// TIA Portal V17 export
// export: Created 2023-02-13T11:16:15.1226472Z, ExportSetting WithDefaults, DisplayName Totally Integrated Automation Portal, DisplayVersion V17, DisplayName TIA Portal Openness, DisplayVersion V17, DisplayName TIA Portal Teamcenter Gateway, DisplayVersion V17, DisplayName TIA Portal Version Control Interface, DisplayVersion V17, DisplayName SINAMICS Startdrive Advanced, DisplayVersion V17, DisplayName SINAMICS Startdrive G130, G150, S120, S150, SINAMICS MV, S210, DisplayVersion V17, DisplayName SINAMICS Startdrive G110M, G120, G120C, G120D, G120P, G115D, DisplayVersion V17, DisplayName STEP 7 Professional, DisplayVersion V17, DisplayName STEP 7 Safety, DisplayVersion V17, DisplayName WinCC Professional, DisplayVersion V17
DATA_BLOCK "IO Valve Homomixer_DB"   // DB4
VERSION : 0.1
// stored: AutoNumber true, DBAccessibleFromOPCUA true, DBAccessibleFromWebserver true, InstanceOfName IO Valve Homomixer, InstanceOfType FB
"IO Valve Homomixer"
   // VAR_INPUT
   //    lock : Bool;
   //    Init : Bool;
   //    testing : Bool;
   //    Reset : Bool;
   // END_VAR
   // VAR
   //    "AV-12.01" { S7_SetPoint := 'True'} : "Valve";
   //    "AV-12.02" { S7_SetPoint := 'True'} : "Valve";
   //    "AV-12.03" { S7_SetPoint := 'True'} : "Valve";
   //    "AV-12.04" { S7_SetPoint := 'True'} : "Valve";
   //    "AV-12.05" { S7_SetPoint := 'True'} : "Valve";
   //    "AV-12.06" { S7_SetPoint := 'True'} : "Valve";
   //    "AV-12.07" { S7_SetPoint := 'True'} : "Valve";
   //    "AV-12.11" { S7_SetPoint := 'True'} : "Valve";
   //    "AV-12.12" { S7_SetPoint := 'True'} : "Valve";
   //    "AV-13.01" { S7_SetPoint := 'True'} : "Valve";
   //    "AV-13.02" { S7_SetPoint := 'True'} : "Valve";
   //    "AV-13.03" { S7_SetPoint := 'True'} : "Valve";
   //    "AV-13.04" { S7_SetPoint := 'True'} : "Valve";
   //    "AV-13.05" { S7_SetPoint := 'True'} : "Valve";
   //    "AV-13.06" { S7_SetPoint := 'True'} : "Valve";
   //    "AV-13.07" { S7_SetPoint := 'True'} : "Valve";
   //    "AV-14.01" { S7_SetPoint := 'True'} : "Valve";
   //    "AV-14.02" { S7_SetPoint := 'True'} : "Valve";
   //    "AV-14.03" { S7_SetPoint := 'True'} : "Valve";
   //    "AV-14.04" { S7_SetPoint := 'True'} : "Valve";
   //    "AV-14.05" { S7_SetPoint := 'True'} : "Valve";
   //    "AV-14.06" { S7_SetPoint := 'True'} : "Valve";
   //    "AV-14.07" { S7_SetPoint := 'True'} : "Valve";
   //    "P-12.01" { S7_SetPoint := 'True'} : "Motor";
   //    "P-13.01" { S7_SetPoint := 'True'} : "Motor";
   //    "P-14.01" { S7_SetPoint := 'True'} : "Motor";
   // END_VAR
BEGIN
END_DATA_BLOCK
